FUNCTION_BLOCK Stamp EXTENDS BaseComponent
VAR_INPUT
END_VAR
VAR_OUTPUT
END_VAR
VAR
	m_stampingCylinder: MonostableCylinder;
	m_slidingCylinder: BistableCylinder;
	m_pressureValve: PropotionalValve;
	
	m_presenceSensor: PresenceSensor;
	m_pressureSensor: PressureSensor;
END_VAR

PROPERTY StampPressure : INT
GET
StampPressure:=m_pressureSensor.Value;
END_GET
SET
m_pressureValve.Pressure := StampPressure;
END_SET
END_PROPERTY

PROPERTY WPAtStart : BOOL
GET
WPAtStart := m_presenceSensor.Value;
END_GET
END_PROPERTY

END_FUNCTION_BLOCK

(* stored: Version 1.1.0.1, ProductVersion 3.1.4024.9
   POU Stamp: Id {d6949c2e-550c-4398-bc8f-e66a02be65d4}, SpecialFunc None
   Property StampPressure: Id {1ebe4f4b-21f1-4fdf-b65b-b6a8dd6044e5}
   Get Get: Id {72a32743-39fb-429d-82c0-0dac5bee17db}
   Set Set: Id {2e7072f7-a7bc-4487-bfb2-ba0c59de3d20}
   Property WPAtStart: Id {e452cfd2-8d5c-43b0-ba65-aca2ebba258c}
   Get Get: Id {1bbd8ce7-30e1-40b3-a618-24dd9b49e9b1} *)
